PROGRAM OP_BTN
VAR
	Start_btn	: BOOL;
	Start_lamp	: BOOL;
	Reset_btn	: BOOL;
	Reset_lamp	: BOOL;
	Estop_btn	: BOOL;
	Estop_lamp	: BOOL;
END_VAR

// Lamp Operation 

Start_lamp := Start_btn AND NOT Reset_btn AND NOT Estop_btn;

Estop_lamp := Estop_btn AND NOT Reset_btn;


// Lamp Reset
IF Reset_btn THEN
	Start_btn := Estop_btn := FALSE;
	Reset_lamp := TRUE;
END_IF

IF Estop_btn THEN
	Start_btn := Reset_btn := FALSE;
	Reset_lamp := FALSE;
END_IF

END_PROGRAM

(* stored: Version 1.1.0.1, ProductVersion 3.1.4024.12
   POU OP_BTN: Id {6774c3e2-553e-4c84-a2e4-62f74f30ccd9}, SpecialFunc None *)
